// Mitsubishi GX Works2 project: 실린더 제어하기 0919   PLC: Q03UDV

PROGRAM MAIN
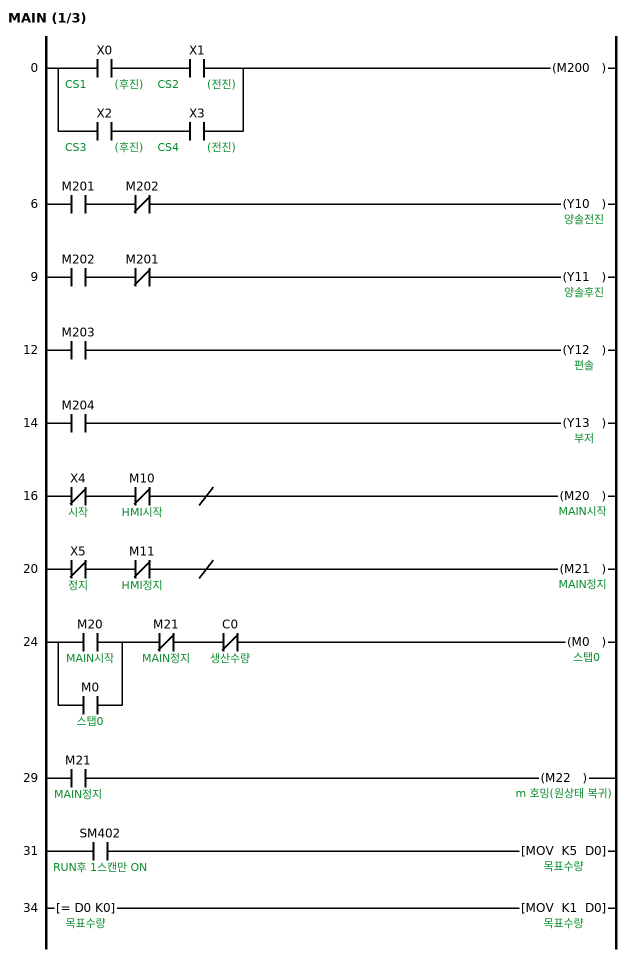
0     LD      X0  ; CS1        (후진)
      AND     X1  ; CS2        (전진)
      LD      X2  ; CS3        (후진)
      AND     X3  ; CS4        (전진)
      ORB
      OUT     M200
6     LD      M201
      ANI     M202
      OUT     Y10  ; 양솔전진
9     LD      M202
      ANI     M201
      OUT     Y11  ; 양솔후진
12    LD      M203
      OUT     Y12  ; 편솔
14    LD      M204
      OUT     Y13  ; 부저
16    LDI     X4  ; 시작
      ANI     M10  ; HMI시작
      INV
      OUT     M20  ; MAIN시작
20    LDI     X5  ; 정지
      ANI     M11  ; HMI정지
      INV
      OUT     M21  ; MAIN정지
24    LD      M20  ; MAIN시작
      OR      M0  ; 스탭0
      ANI     M21  ; MAIN정지
      ANI     C0  ; 생산수량
      OUT     M0  ; 스탭0
29    LD      M21  ; MAIN정지
      OUT     M22  ; m 호밍(원상태 복귀)
31    LD      SM402  ; RUN후 1스캔만 ON
      MOV     K5 D0  ; 목표수량
34    LD=     D0 K0  ; 목표수량
      MOV     K1 D0
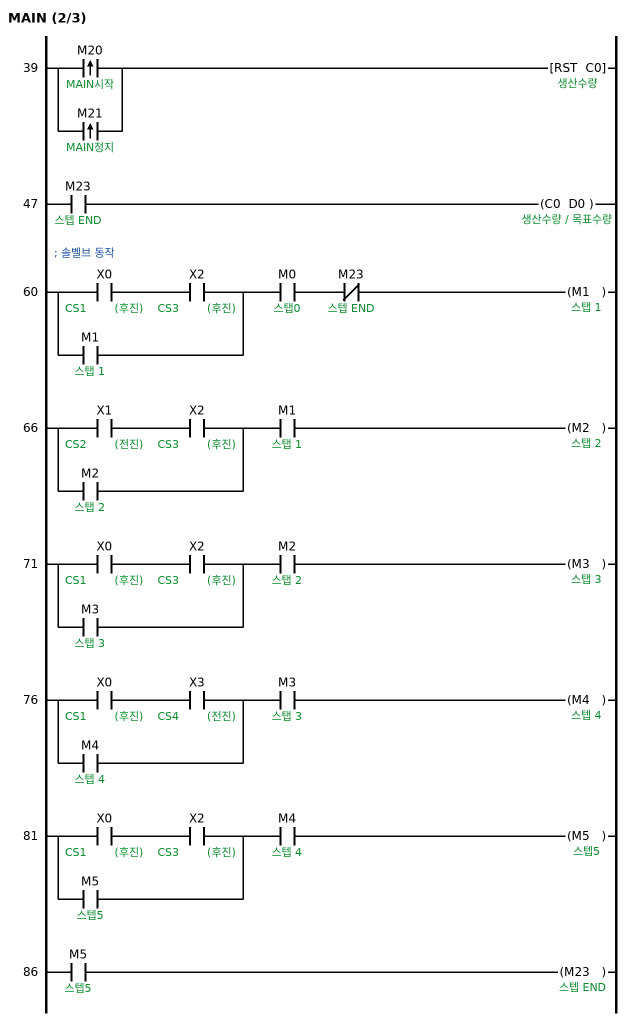
39    LDP     M20  ; MAIN시작
      ORP     M21  ; MAIN정지
      RST     C0  ; 생산수량
47    LD      M23  ; 스텝 END
      OUT     C0 D0  ; 생산수량 / 목표수량
; 솔벨브 동작
60    LD      X0  ; CS1        (후진)
      AND     X2  ; CS3        (후진)
      OR      M1  ; 스탭 1
      AND     M0  ; 스탭0
      ANI     M23  ; 스텝 END
      OUT     M1  ; 스탭 1
66    LD      X1  ; CS2        (전진)
      AND     X2  ; CS3        (후진)
      OR      M2  ; 스탭 2
      AND     M1  ; 스탭 1
      OUT     M2  ; 스탭 2
71    LD      X0  ; CS1        (후진)
      AND     X2  ; CS3        (후진)
      OR      M3  ; 스탭 3
      AND     M2  ; 스탭 2
      OUT     M3  ; 스탭 3
76    LD      X0  ; CS1        (후진)
      AND     X3  ; CS4        (전진)
      OR      M4  ; 스텝 4
      AND     M3  ; 스탭 3
      OUT     M4  ; 스텝 4
81    LD      X0  ; CS1        (후진)
      AND     X2  ; CS3        (후진)
      OR      M5  ; 스텝5
      AND     M4  ; 스텝 4
      OUT     M5  ; 스텝5
86    LD      M5  ; 스텝5
      OUT     M23  ; 스텝 END
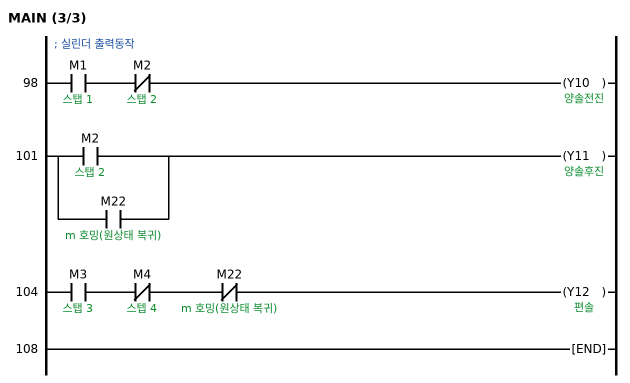
; 실린더 출력동작
98    LD      M1  ; 스탭 1
      ANI     M2  ; 스탭 2
      OUT     Y10  ; 양솔전진
101   LD      M2  ; 스탭 2
      OR      M22  ; m 호밍(원상태 복귀)
      OUT     Y11  ; 양솔후진
104   LD      M3  ; 스탭 3
      ANI     M4  ; 스텝 4
      ANI     M22  ; m 호밍(원상태 복귀)
      OUT     Y12  ; 편솔
108   END
END_PROGRAM
